FUNCTION_BLOCK FB_HardwareOutputs


;
// Example
(*
Q_11_001_SG := fbSG_001.HW_Outputs;
Q_11_001_SG_Beacon_Error := fbSG_001.HW_Outputs.ErrorPending;
Q_11_001_SG_Beacon_Auto := fbSG_001.HW_Outputs.GroupStarted;
*)

END_FUNCTION_BLOCK

(* stored: Version 1.1.0.1, ProductVersion 3.1.4024.9
   POU FB_HardwareOutputs: Id {ec90984b-3be2-403d-a066-1c53f5f3e002}, SpecialFunc None *)
